Fanuc TP program (LS listing): OP10_1_CLS_CHUCK.LS

/PROG  OP10_1_CLS_CHUCK
/ATTR
OWNER		= MNEDITOR;
COMMENT		= "CHUCK CLOSE";
PROG_SIZE	= 525;
CREATE		= DATE 17-09-25  TIME 18:00:38;
MODIFIED	= DATE 17-09-29  TIME 16:21:44;
FILE_NAME	= M1_ORIEN;
VERSION		= 0;
LINE_COUNT	= 18;
MEMORY_SIZE	= 997;
PROTECT		= READ;
TCD:  STACK_SIZE	= 0,
      TASK_PRIORITY	= 50,
      TIME_SLICE	= 0,
      BUSY_LAMP_OFF	= 0,
      ABORT_REQUEST	= 0,
      PAUSE_REQUEST	= 0;
DEFAULT_GROUP	= *,*,*,*,*;
CONTROL_CODE	= 00000000 00000000;
/APPL

AUTO_SINGULARITY_HEADER;
  ENABLE_SINGULARITY_AVOIDANCE   : TRUE;
/MN
   1:  LBL[1:START] ;
   2:  $WAITTMOUT=400 ;
   3:  R[43:ACTION RETRIES]=0    ;
   4:   ;
   5:  LBL[100:CLOSE CHUCK] ;
   6:  R[43:ACTION RETRIES]=R[43:ACTION RETRIES]+1    ;
   7:  IF R[43:ACTION RETRIES]>=3,JMP LBL[9990] ;
   8:  DO[135:OFF:OP10R-1 CHUCK CLOSE]=PULSE,0.5sec ;
   9:  WAIT DI[135:OFF:OP10R-1 CHUCK CLOSED]=ON TIMEOUT,LBL[100] ;
  10:  JMP LBL[9999] ;
  11:   ;
  12:  LBL[9990:CHUCK FAULT] ;
  13:  CALL CHUCK_MSG(3) ;
  14:  UALM[6] ;
  15:  R[43:ACTION RETRIES]=0    ;
  16:  JMP LBL[1] ;
  17:   ;
  18:  LBL[9999:END] ;
/POS
/END
